{attribute 'linkalways'} 
{attribute 'no_explicit_call' := 'This FB is a CLASS and must be accessed using methods or properties'}
{attribute 'enable_dynamic_creation'}
FUNCTION_BLOCK Node_ContainerType_Vector_TcVnRotatedRectangle EXTENDS Node
VAR
    out : _GUID;
END_VAR

METHOD PUBLIC  Clone : I_Node
VAR
	pNode : POINTER TO Node_ContainerType_Vector_TcVnRotatedRectangle;
END_VAR
pNode := __NEW(Node_ContainerType_Vector_TcVnRotatedRectangle);
Clone := pNode^;
END_METHOD

METHOD FB_init : BOOL
VAR_INPUT
	bInitRetains : BOOL; // if TRUE, the retain variables are initialized (warm start / cold start)
	bInCopyCode : BOOL;  // if TRUE, the instance afterwards gets moved into the copy code (online change)
END_VAR
AddOutput('out', out);
END_METHOD

METHOD PROTECTED OnExecute
out.Value := ContainerType_Vector_TcVnRotatedRectangle;
END_METHOD

END_FUNCTION_BLOCK

(* stored: Version 1.1.0.1, ProductVersion 3.1.4026.17
   POU Node_ContainerType_Vector_TcVnRotatedRectangle: Id {b0bbd9f2-298a-0cf5-224b-bee25340b558}, SpecialFunc None
   Folder Constructor: Id {58f27be7-69f9-0dd2-1d69-92bc89afcdbd}
   Method Clone: Id {07491e13-cda9-0c1f-2cf5-f13c88d9cb12}
   Method FB_init: Id {e7ca3b11-bfe0-0171-2070-91dcdea55c24}
   Method OnExecute: Id {00e107b6-643e-0cf5-1a20-9a08ab155471} *)
